Staubli VAL3: master5.pjx

--- master5.pjx ---
Parameters version=s7.7.2 stackSize=5000 millimeterUnit=true
Program file=start.pgx
Program file=stop.pgx
Data file=master5.dtx

--- master5.dtx ---
public frame fUserFrame = {fatherId=world[0]}
public jointRx jtPark = {j1=-90, j2=-20, j3=140, j5=-60, j6=178}
public jointRx ptRoutingPath = {j1=10.546, j2=44.21, j3=63.432, j4=13.525, j5=70.04, j6=120.724}
public mdesc mNomSpeed = {blend=off}
public mdesc mdJointBlend = {accel=250, decel=150, leave=1, reach=1}
public mdesc mdLineBlend = {accel=80, vel=60, decel=50, rmax=9999, tmax=100, leave=2, reach=2}
public tool tTool = {x=485, y=70, z=-90.5, rx=5, rz=-92.998, fatherId=flange[0], ioLink=valve1}
